// Mitsubishi GX Works2 project: SEGUNDO EJERCICIO   PLC: FX0S/FX0

PROGRAM MAIN
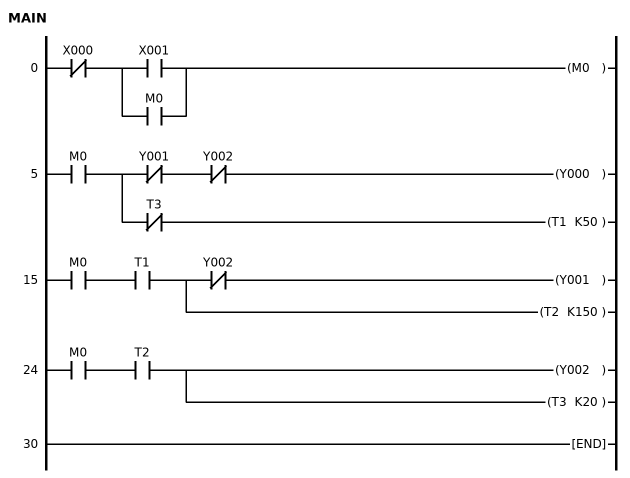
0     LDI     X000
      LD      X001
      OR      M0
      ANB
      OUT     M0
5     LD      M0
      MPS
      ANI     Y001
      ANI     Y002
      OUT     Y000
      MPP
      ANI     T3
      OUT     T1 K50
15    LD      M0
      AND     T1
      MPS
      ANI     Y002
      OUT     Y001
      MPP
      OUT     T2 K150
24    LD      M0
      AND     T2
      OUT     Y002
      OUT     T3 K20
30    END
END_PROGRAM
